(* Schneider Machine Expert - Basic project SAU4, file version 2.0.0.0 *)
(* ProjectInformations: Name=New project *)

HARDWARE
  Cpu 0: TM221CE16T
  Cartridge1 0: TMC2SL1
  EthernetConfiguration: NetworkName=M221, IpAllocationMode=FixedAddress, IpAddress=192.168.1.14, SubnetMask=255.255.255.0
  EthernetConfiguration: NetworkName=M221, IpAllocationMode=FixedAddress, IpAddress=0.0.0.0, SubnetMask=0.0.0.0
  SerialLineConfiguration: Baud=Baud9600, Parity=ParityNone, DataBits=DataBits8, StopBits=StopBits1, PhysicalMedium=PhysicalMediumRs485, TransmissionMode=TransmissionModeModbusRtu, SlaveId=1, Addressing=MasterAddressing
  MastTask: UsePeriodScanMode=false, PeriodScan=100
  FastTask: Period=255
  CpuBehavior: StartingMode=StartAsPreviousState, AutoSaveRamOnEeprom=true, WatchdogPeriod=250

SYMBOLS  (address, symbol, comment, settings)
  %S5       SB_TB100MS  "内部时钟生成的 100 毫秒时基"
  %TM0        [Preset=15, Base=OneSecond]
  %TM1        [Preset=10, Base=TenMilliSeconds]
  %TM2        [Preset=15, Base=OneSecond]
  %READ_VAR0   [Link(Value(FBComLinkParameterEnums=SerialLine1)), RemoteDeviceId(Value(int=1)), Timeout(Value(int=3)), ObjType(Value(FBComObjTypeParameterEnums=IW)), FirstObj(Value(int=513)), Quantity(Value(int=2)), IndexData(Value(int=0))]
  %READ_VAR1   [Link(Value(FBComLinkParameterEnums=SerialLine1)), RemoteDeviceId(Value(int=2)), Timeout(Value(int=3)), ObjType(Value(FBComObjTypeParameterEnums=IW)), FirstObj(Value(int=513)), Quantity(Value(int=8)), IndexData(Value(int=10))]

POU Communication
  (* SectionNumber=0 *)

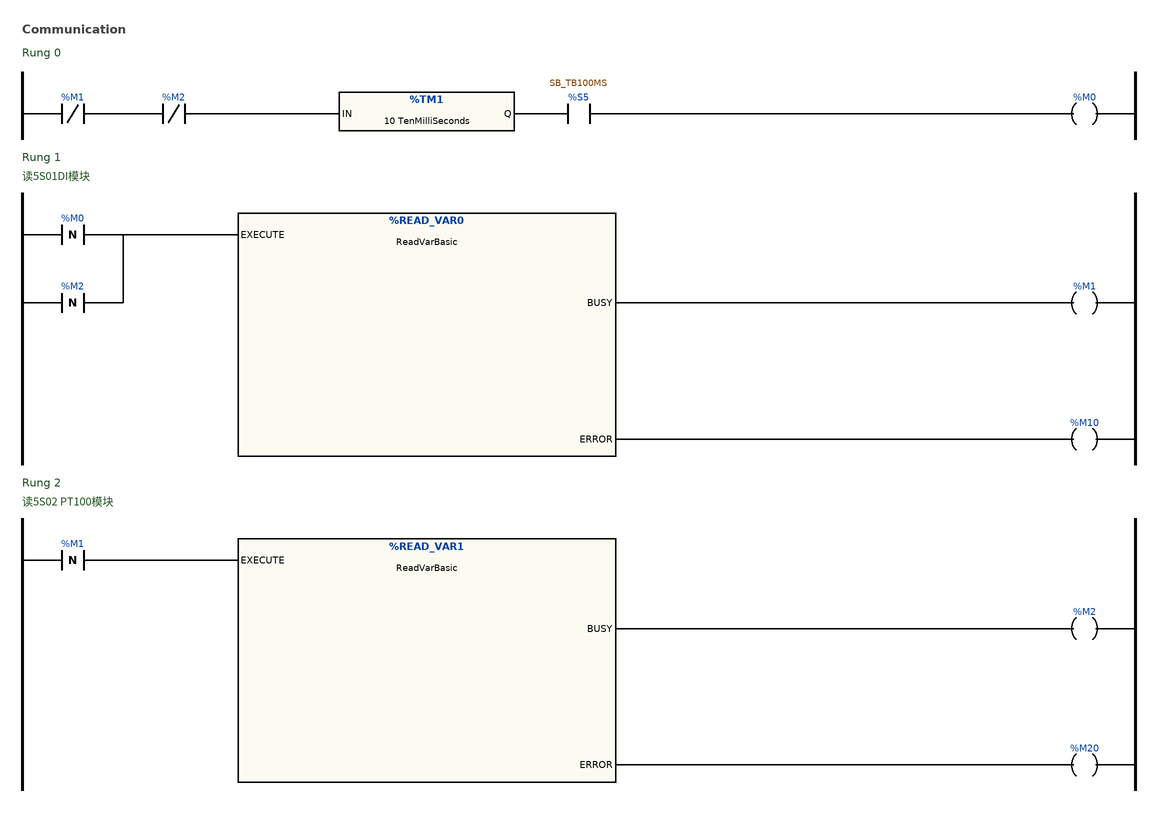

// Rung 0
  BLK %TM1
  LDN %M1
  ANDN %M2
  IN
  OUT_BLK
  LD Q
  AND %S5                 (* SB_TB100MS *)
  ST %M0
  END_BLK
  // as ST:
  //   %TM1(IN := NOT %M1 AND NOT %M2);
  //   %M0 := %TM1.Q AND SB_TB100MS;

// Rung 1
// 读5S01DI模块
  BLK %READ_VAR0
  LDF %M0
  ORF %M2
  EXECUTE
  OUT_BLK
  LD BUSY
  ST %M1
  LD ERROR
  ST %M10
  END_BLK
  // as ST:
  //   %READ_VAR0(EXECUTE := FALLING(%M0) OR FALLING(%M2));
  //   %M1 := %READ_VAR0.BUSY;
  //   %M10 := %READ_VAR0.ERROR;

// Rung 2
// 读5S02 PT100模块
  BLK %READ_VAR1
  LDF %M1
  EXECUTE
  OUT_BLK
  LD BUSY
  ST %M2
  LD ERROR
  ST %M20
  END_BLK
  // as ST:
  //   %READ_VAR1(EXECUTE := FALLING(%M1));
  //   %M2 := %READ_VAR1.BUSY;
  //   %M20 := %READ_VAR1.ERROR;

POU CommError
  (* SectionNumber=0 *)

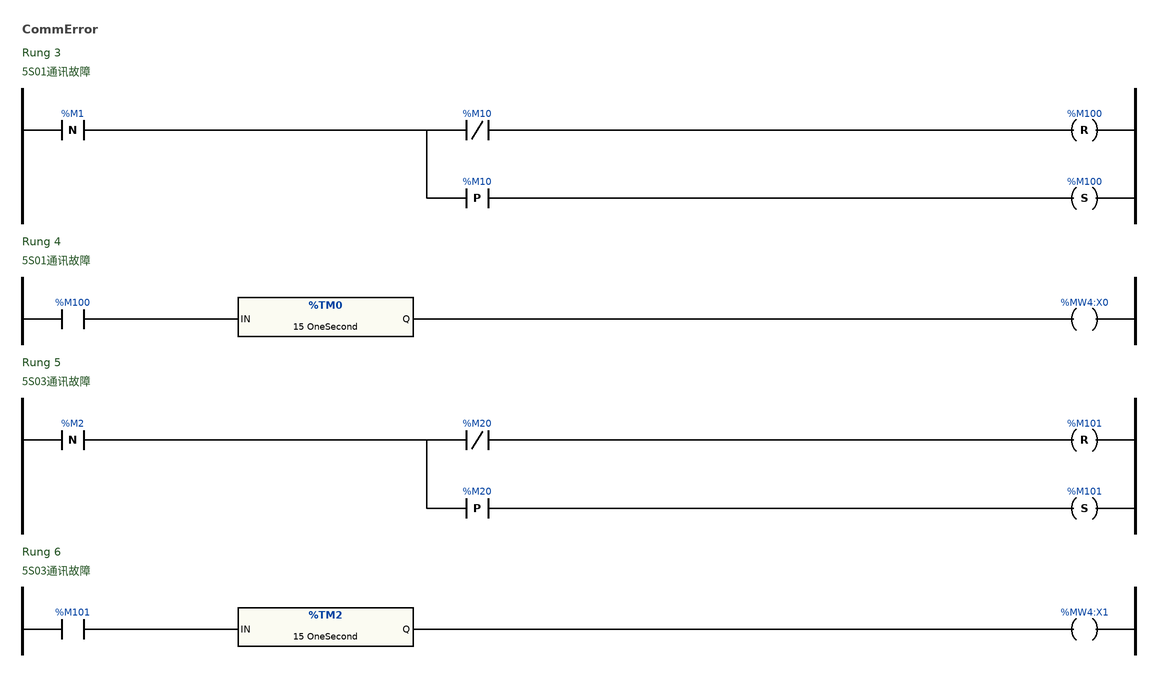

// Rung 3
// 5S01通讯故障
  LDF %M1
  MPS
  ANDN %M10
  R %M100
  MPP
  ANDR %M10
  S %M100
  // as ST:
  //   IF FALLING(%M1) AND NOT %M10 THEN %M100 := FALSE; END_IF;
  //   IF FALLING(%M1) AND RISING(%M10) THEN %M100 := TRUE; END_IF;

// Rung 4
// 5S01通讯故障
  BLK %TM0
  LD %M100
  IN
  OUT_BLK
  LD Q
  ST %MW4:X0
  END_BLK
  // as ST:
  //   %TM0(IN := %M100);
  //   %MW4:X0 := %TM0.Q;

// Rung 5
// 5S03通讯故障
  LDF %M2
  MPS
  ANDN %M20
  R %M101
  MPP
  ANDR %M20
  S %M101
  // as ST:
  //   IF FALLING(%M2) AND NOT %M20 THEN %M101 := FALSE; END_IF;
  //   IF FALLING(%M2) AND RISING(%M20) THEN %M101 := TRUE; END_IF;

// Rung 6
// 5S03通讯故障
  BLK %TM2
  LD %M101
  IN
  OUT_BLK
  LD Q
  ST %MW4:X1
  END_BLK
  // as ST:
  //   %TM2(IN := %M101);
  //   %MW4:X1 := %TM2.Q;
